INTERFACE I_Gripper

END_INTERFACE

(* stored: Version 1.1.0.1, ProductVersion 3.1.4024.12
   Itf I_Gripper: Id {e1d98384-a7fe-4388-bdfe-d750f3fbb218} *)
